// TIA Portal V21 export
VAR_GLOBAL   // PLC tag table "K_AzionamentoFesto_CMMT-ST"
END_VAR
VAR_GLOBAL CONSTANT   // user constants
   "K_AzionamentoFesto_CMMT-ST_AltezzaStampo" : Int := 1;
END_VAR
